(* IEC 61131-3 sources: Industry-PLC-LLM/data/PLCBEAD_repo/PLCBEAD_PLCEmbed-main/PLC-BEAD/Source/GEB/F_TO_C, 1 file *)

(* ---- F_TO_C.ST ---- *)
FUNCTION F_TO_C:REAL
	VAR_INPUT
		FAHRENHEIT :	REAL;
	END_VAR
	F_TO_C := (FAHRENHEIT - 32.0) * 0.5555555555555;
END_FUNCTION

PROGRAM program0
  VAR
    LocalVar0 : REAL;
	LocalOUT  : REAL;
  END_VAR
  	LocalOUT := F_TO_C(LocalVar0);
END_PROGRAM
